FUNCTION_BLOCK M_SUB (* Subtract two matrices of REAL *)
  (* Standard: 61499-1; Classification: Matrix Operations; Function: Addition *)
  (* Version 0.1, 2007-10-19, JHC, Holobloc Inc, Moved to fb.rt.math.matrix. *)
  (* Version 0.0, 2002-03-06, JHC, Rockwell Automation *)
  (* Compiler header: package fb.rt.math.matrix; *)
  (* Compiler Java IBM VisualAge 3.0 *)
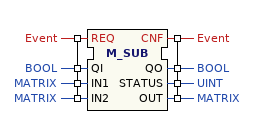
  EVENT_INPUT
    REQ WITH QI, IN1, IN2; (* Set OUT to IN1-IN2 *)
  END_EVENT
  EVENT_OUTPUT
    CNF WITH QO, STATUS, OUT; (* Confirmation of Requested Service *)
  END_EVENT
  VAR_INPUT
    QI : BOOL; (* Event Input Qualifier *)
    IN1 : MATRIX; (* Minuend *)
    IN2 : MATRIX; (* Subtrahend *)
  END_VAR
  VAR_OUTPUT
    QO : BOOL; (* Event Output Qualifier *)
    STATUS : UINT; (* Service Status *)
    OUT : MATRIX; (* Difference *)
  END_VAR
END_FUNCTION_BLOCK
